INTERFACE I_BOOL EXTENDS I_Datatype

PROPERTY PUBLIC Value : REFERENCE TO BOOL
GET
END_GET
END_PROPERTY

END_INTERFACE

(* stored: Version 1.1.0.1, ProductVersion 3.1.4024.15
   Itf I_BOOL: Id {2d62b881-0911-0444-1cdc-0d16292885b7}
   Property Value: Id {d3b10817-168c-0d7a-17cb-d166ae80aef6}
   Get Get: Id {e70f7280-1da4-042e-250c-714a07de0e95} *)
